Universal Robots PolyScope program: orange_Bridge_flat_roof.urp

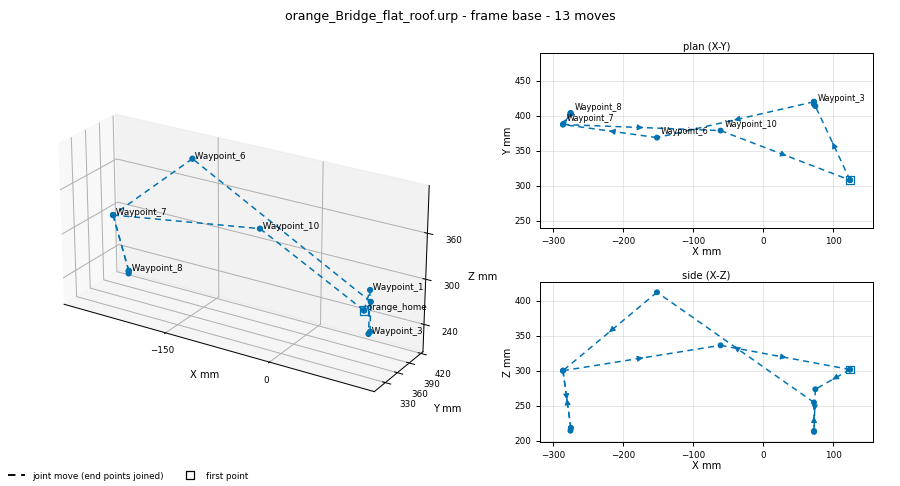
[picture p0: tool path of orange_Bridge_flat_roof.urp in frame base, 13 of 13 moves have a stored position in this frame; points joined in program order, loops and branches not executed]
Program orange_Bridge_flat_roof (installation=default directory=/programs/usbdisk/Zahra1/orangi createdIn=5.11.11.1010533 lastSavedIn=5.11.11.1010533 robotSerialNumber=20205300864)
Calibrated DH parameters: a=[-0.000166, -0.243494, -0.153108, 0.000057, -0.000123, 0]; d=[0.151897, -1.34267, 53.988124, -52.514559, 0.085283, 0.092193]; alpha=[1.572472, -0.003756, 0.002824, 1.570807, -1.572621, 0]; deltaTheta=[0, 0.020704, 7.033215, -0.770746, 0.000004, 0]
Robot Program (runOnlyOnce=true)
  MoveJ speed 60 deg/s, acceleration 80 deg/s^2 (useActiveTCP=true) feature=Base
    Waypoint orange_home: TCP in base x=124.286 y=308.277 z=301.462 mm, rx=2.2499 ry=-2.1846 rz=-0.0963 rad; joints [-269.66, -91.226, -90.279, -86.086, 92.69, 808.818] deg
    Waypoint Waypoint_1: TCP in base x=74.759 y=413.974 z=273.278 mm, rx=2.2395 ry=-2.1514 rz=-0.0559 rad; joints [-262.835, -114.841, -67.338, -87.391, 92.822, 814.969] deg
    URCap Gripper (Robotiq_Grippers, Robotiq Inc.) dataModel(position=27.84313725490196, force=94.0, speed=40.0, positionInDouble=27.84313725490196, forceInDouble=94.0, speedInDouble=40.0, slaveIds=[9], blocking=true, robotCompliant=false)
    Waypoint Waypoint_3: TCP in base x=72.866 y=416.362 z=212.478 mm, rx=2.1592 ry=-2.2297 rz=-0.0375 rad; joints [-262.562, -117.96, -79.009, -73.095, 92.504, 819.399] deg
    URCap Gripper (Robotiq_Grippers, Robotiq Inc.) dataModel(position=58.549019607843135, force=94.0, speed=40.0, positionInDouble=58.549019607843135, forceInDouble=94.0, speedInDouble=40.0, slaveIds=[9], blocking=true, robotCompliant=false)
    Waypoint Waypoint_4: TCP in base x=72.851 y=420.085 z=213.8 mm, rx=2.164 ry=-2.2139 rz=-0.0227 rad; joints [-262.635, -118.962, -76.766, -75.066, 92.545, 818.769] deg
    Waypoint Waypoint_5: TCP in base x=72.825 y=420.078 z=254.425 mm, rx=2.164 ry=-2.2137 rz=-0.0226 rad; joints [-262.613, -117.107, -68.515, -85.179, 92.536, 818.765] deg
    Waypoint Waypoint_6: TCP in base x=-151.236 y=368.905 z=411.753 mm, rx=-2.1806 ry=2.2432 rz=0.0888 rad; joints [-228.359, -119.938, -20.415, -126.264, 89.278, 853.262] deg
    Waypoint Waypoint_7: TCP in base x=-285.477 y=387.647 z=299.823 mm, rx=2.1235 ry=-2.2977 rz=-0.0367 rad; joints [-217.941, -135.422, -26.231, -106.799, 90.325, 866.586] deg
    Waypoint Waypoint_8: TCP in base x=-274.22 y=403.585 z=218.07 mm, rx=2.1561 ry=-2.2207 rz=-0.0686 rad; joints [-220.756, -134.017, -51.637, -81.476, 92.257, 861.05] deg
    Waypoint Waypoint_2: TCP in base x=-274.796 y=404.102 z=214.129 mm, rx=2.1579 ry=-2.2225 rz=-0.0594 rad; joints [-220.739, -134.503, -51.675, -81.305, 92.155, 861.056] deg
    URCap Gripper (Robotiq_Grippers, Robotiq Inc.) dataModel(position=25.098039215686274, force=94.0, speed=40.0, positionInDouble=25.098039215686274, forceInDouble=94.0, speedInDouble=40.0, slaveIds=[9], blocking=true, robotCompliant=false)
    Waypoint Waypoint_8: TCP in base x=-274.22 y=403.585 z=218.07 mm, rx=2.1561 ry=-2.2207 rz=-0.0686 rad; joints [-220.756, -134.017, -51.637, -81.476, 92.257, 861.05] deg
    Waypoint Waypoint_7: TCP in base x=-285.477 y=387.647 z=299.823 mm, rx=2.1235 ry=-2.2977 rz=-0.0367 rad; joints [-217.941, -135.422, -26.231, -106.799, 90.325, 866.586] deg
    Waypoint Waypoint_10: TCP in base x=-60.503 y=378.951 z=335.988 mm, rx=-2.2043 ry=2.0992 rz=0.031 rad; joints [-239.746, -103.735, -66.779, -96.708, 84.912, 837.407] deg
    Waypoint orange_home: TCP in base x=124.286 y=308.277 z=301.462 mm, rx=2.2499 ry=-2.1846 rz=-0.0963 rad; joints [-269.66, -91.226, -90.279, -86.086, 92.69, 808.818] deg
